Staubli VAL3: start.pgx

program start()
  local bool l_bRes
begin

     call TxtFile:ReadAction(l_bRes)
  if !l_bRes
    popUpMsg("读取动作文件出错")
    return
  endIf
    call TxtFile:ReadPreset(l_bRes)
  if !l_bRes
    popUpMsg("读取工艺文件出错")
    return
  endIf
  call TxtFile:ReadProductName("Disk://Txt/Recipe.txt",l_bRes)
   if !l_bRes
    popUpMsg("读取生产文件出错")
    return
  endIf
call TxtFile:ReadProduct("Disk://Txt/Recipe.txt",TxtFile:sProductName,true,l_bRes)
   if !l_bRes
    popUpMsg("读取生产文件出错")
    return
  endIf


 nStartTraj=1
 nEndTraj=TxtFile:nTotalTraj
 taskCreate "ReadFile",50,ReadTraj()
 taskCreate "Preset",100,Preset()

 call Move()

end
